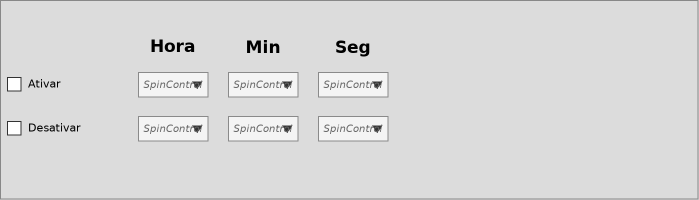
VISUALIZATION ProgramacaoHoraria  // 699x200
VAR_IN_OUT

END_VAR
VAR_INPUT
	uiIndex:UINT;		//Indice da programacao horaria
	wDayOfWeek:WORD;	
END_VAR
    Checkbox (5,69 120x30), "Ativar", variable: GVL_TimeSch.aTimeToSchActivate[wDayOfWeek,uiIndex].bUse
    Checkbox (5,113 120x30), "Desativar", variable: GVL_TimeSch.aTimeToSchDeactivate[wDayOfWeek,uiIndex].bUse
    SpinControl (138,72 70x25), variable: GVL_TimeSch.aTimeToSchActivate[wDayOfWeek,uiIndex].wHour
        OnMouseClick: write the text variable via Default, min 0, max 23
    Label (138,31 70x30), "Hora"
    SpinControl (228,72 70x25), variable: GVL_TimeSch.aTimeToSchActivate[wDayOfWeek,uiIndex].wMinute
        OnMouseClick: write the text variable via Default, min 0, max 59
    Label (228,32 70x30), "Min"
    SpinControl (318,72 70x25), variable: GVL_TimeSch.aTimeToSchActivate[wDayOfWeek,uiIndex].wSecond
        OnMouseClick: write the text variable via Default, min 0, max 59
    Label (318,32 70x30), "Seg"
    SpinControl (138,116 70x25), variable: GVL_TimeSch.aTimeToSchDeactivate[wDayOfWeek,uiIndex].wHour
        OnMouseClick: write the text variable via Default, min 0, max 23
    SpinControl (228,116 70x25), variable: GVL_TimeSch.aTimeToSchDeactivate[wDayOfWeek,uiIndex].wMinute
        OnMouseClick: write the text variable via Default, min 0, max 59
    SpinControl (318,116 70x25), variable: GVL_TimeSch.aTimeToSchDeactivate[wDayOfWeek,uiIndex].wSecond
        OnMouseClick: write the text variable via Default, min 0, max 59
END_VISUALIZATION

(* stored: Version 1.1.0.1
   Visu ProgramacaoHoraria: Id {539c5574-5f47-43d1-9698-634b6716ac0a} *)
